SUBAPPLICATION Uebung_160b2_AX (* Motor Links/Rechtslauf Automatisierung IXA *)
  (* Standard: 61499-2; Description: Copyright (c) 2023 Meisterschulen am Ostbahnhof This program and the accompanying materials are made available under the terms of the Eclipse Public License 2.0 which is available at https://www.eclipse.org/legal/epl-2.0/ SPDX-License-Identifier: EPL-2.0 *)
  (* Version 1.0, 2023-10-23, Franz Höpfinger, Meisterschulen am Ostbahnhof, initial API and implementation and/or initial documentation *)
  PACKAGE Uebungen;
  IMPORT logiBUS::io::DI::logiBUS_DI::Input_I1;
  IMPORT logiBUS::io::DI::logiBUS_DI::Input_I2;
  IMPORT logiBUS::io::DI::logiBUS_DI::Input_I3;
  IMPORT logiBUS::io::DQ::logiBUS_DO::Output_Q5;
  IMPORT logiBUS::io::DQ::logiBUS_DO::Output_Q56;
  IMPORT logiBUS::io::DQ::logiBUS_DO::Output_Q6;
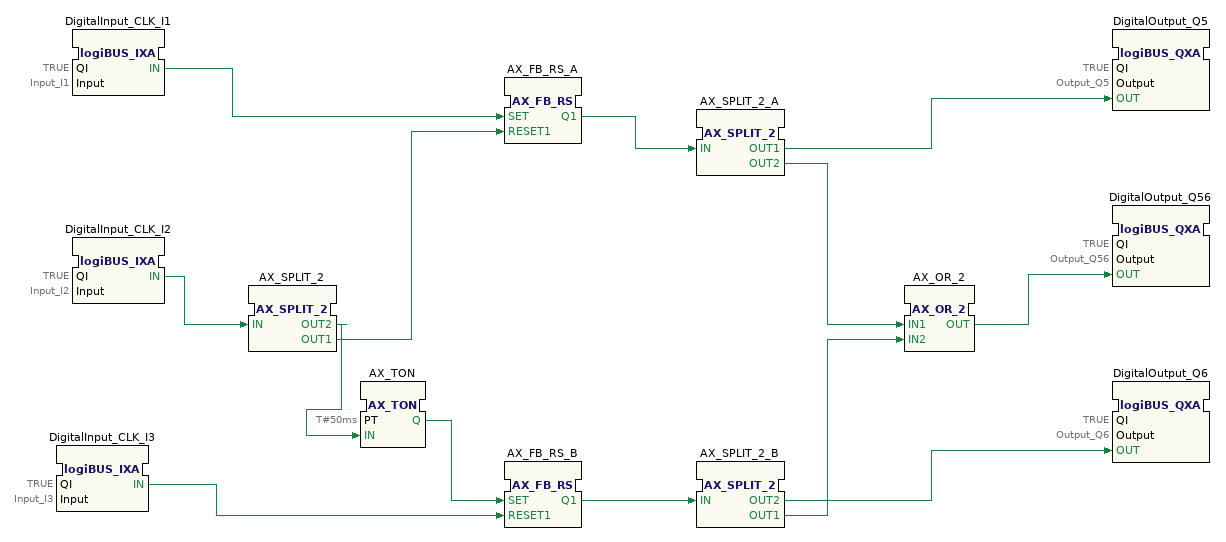
  FBS
    DigitalOutput_Q5 : logiBUS::io::DQ::logiBUS_QXA(QI := TRUE, Output := Output_Q5);
    DigitalOutput_Q6 : logiBUS::io::DQ::logiBUS_QXA(QI := TRUE, Output := Output_Q6);
    AX_OR_2 : adapter::booleanOperators::AX_OR_2;
    DigitalOutput_Q56 : logiBUS::io::DQ::logiBUS_QXA(QI := TRUE, Output := Output_Q56);
    AX_SPLIT_2_A : adapter::events::unidirectional::AX_SPLIT_2;
    AX_SPLIT_2_B : adapter::events::unidirectional::AX_SPLIT_2;
    DigitalInput_CLK_I2 : logiBUS::io::DI::logiBUS_IXA(QI := TRUE, Input := Input_I2);
    DigitalInput_CLK_I1 : logiBUS::io::DI::logiBUS_IXA(QI := TRUE, Input := Input_I1);
    AX_FB_RS_A : adapter::iec61131::bistableElements::AX_FB_RS;
    DigitalInput_CLK_I3 : logiBUS::io::DI::logiBUS_IXA(QI := TRUE, Input := Input_I3);
    AX_FB_RS_B : adapter::iec61131::bistableElements::AX_FB_RS;
    AX_TON : adapter::events::unidirectional::timers::AX_TON(PT := T#50ms);
    AX_SPLIT_2 : adapter::events::unidirectional::AX_SPLIT_2;
  END_FBS
  ADAPTER_CONNECTIONS
    AX_SPLIT_2_A.OUT1 TO DigitalOutput_Q5.OUT;
    AX_SPLIT_2_B.OUT2 TO DigitalOutput_Q6.OUT;
    AX_OR_2.OUT TO DigitalOutput_Q56.OUT;
    AX_SPLIT_2_A.OUT2 TO AX_OR_2.IN1;
    AX_SPLIT_2_B.OUT1 TO AX_OR_2.IN2;
    AX_FB_RS_A.Q1 TO AX_SPLIT_2_A.IN;
    AX_FB_RS_B.Q1 TO AX_SPLIT_2_B.IN;
    DigitalInput_CLK_I1.IN TO AX_FB_RS_A.SET;
    DigitalInput_CLK_I2.IN TO AX_SPLIT_2.IN;
    AX_TON.Q TO AX_FB_RS_B.SET;
    DigitalInput_CLK_I3.IN TO AX_FB_RS_B.RESET1;
    AX_SPLIT_2.OUT2 TO AX_TON.IN;
    AX_SPLIT_2.OUT1 TO AX_FB_RS_A.RESET1;
  END_CONNECTIONS
END_SUBAPPLICATION
